// TIA Portal V20 export
DATA_BLOCK "BK13"   // DB249
// stored: MemoryReserve 100
   VAR
      "X10-1 SPARE" : Bool;
      "X11-1 SPARE" : Bool;
      "X12-1 HP STAGE LIFT #2 FRONT DOWN" : Bool;
      "X13-1 HP STAGE LIFT #2 REAR DOWN" : Bool;
      "X14-1 HP STACK DETECT SENSOR 2" : Bool;
      "X15-1 HP STAGE 2 SAFETY PIN LOADING SENSOR" : Bool;
      "X16-1 SPARE" : Bool;
      "X17-1 THICKNESS TEST SENSOR AMP POWER" : Bool;
      "X10-2 SPARE" : Bool;
      "X11-2 SPARE" : Bool;
      "X12-2 HP STAGE LIFT #2 FRONT UP" : Bool;
      "X13-2 HP STAGE LIFT #2 REAR UP" : Bool;
      "X14-2 SPARE" : Bool;
      "X15-2 SPARE" : Bool;
      "X16-2 SPARE" : Bool;
      "X17-2 SPARE" : Bool;
   END_VAR
BEGIN
END_DATA_BLOCK
